(* CoDeSys 2.3 library: 3000ext.lib *)

(* Global variable list: Global_Constants *)
VAR_GLOBAL CONSTANT
(*CAN buses*)
	G_CANAPI_CAN1:BYTE := 0;
	G_CANAPI_CAN2:BYTE := 1;

(*Configuration flags*)
  	G_CANAPI_CFG_FLAGS_LISTEN_ONLY:WORD:=		16#0004;	(*CAN-interface is set to listen only mode*)

(*bit rates*)
	G_CANAPI_BAUDRATE_10K:WORD:= 	10;
	G_CANAPI_BAUDRATE_20K:WORD:= 	20;
	G_CANAPI_BAUDRATE_50K:WORD:= 	50;
	G_CANAPI_BAUDRATE_125K:WORD:= 	125;
	G_CANAPI_BAUDRATE_250K:WORD:= 	250;
	G_CANAPI_BAUDRATE_500K:WORD:= 	500;
	G_CANAPI_BAUDRATE_800K:WORD:= 	800;
	G_CANAPI_BAUDRATE_1000K:WORD:=1000;

(*protocols*)
	G_CANAPI_PROTOCOL_CANOPEN:BYTE := 0;
	G_CANAPI_PROTOCOL_ISOBUS:BYTE := 1;

END_VAR

(* Data type *)
TYPE CanApiBusConfiguration :
STRUCT
	i_enabled:WORD;			(* Used only internally. Variable is not needed in		*)
							(* function call CANAPI_INIT_BUS.						*)
	i_nbrOfInterface:WORD;	(* Number of the CAN channel channel(0,1,..)			*)
	i_bitRate:WORD;			(* CAN bitrate 											*)
	i_configFlags:WORD;		(* Configuration flags. See global contants				*)
END_STRUCT
END_TYPE

(* Data type *)
TYPE CanApiBusTimingParameters :
STRUCT
	i_nominalBitRate:DWORD;	(* CAN bitrate *)
	i_propSegment:WORD;		(* Propagation time segment (Tprop) *)
	i_phaseSegment1:WORD;	(* Phase buffer segment 1 (Tb1) *)
	i_phaseSegment2:WORD;	(* Phase buffer segment 2 (Tb2) *)
	i_sjw:WORD;					(* Resynchronization jump width (Tsjw) *)
	i_bitRateTolerance:WORD;	(*Allowed error in calculated bitRate.
									   Value in passed in 0.1 percent. So i.e. 15 means 1,5% *)
END_STRUCT
END_TYPE

(* Data type *)
TYPE CanApiMessage :
STRUCT
	id		: DWORD;				(*COB-ID of the message*)
	msgData	: ARRAY[0..7] OF BYTE;	(*Message data*)
	len		: BYTE;					(*Length of the message*)
END_STRUCT
END_TYPE

(* Data type *)
TYPE CanApiStatus :
STRUCT
	busOffCount		: DWORD;	(* Bus-Off error count *)
    ewarnCount		: DWORD;	(* EWarn Count *)

	txFifoOverruns	: DWORD;	(* Tx fifo overrun count *)
	txCount			: DWORD;	(* Tx message count *)
	txErrors		: DWORD;	(* Tx error count *)

	rxCount			: DWORD;	(* Rx message count *)
	rxErrors		: DWORD;   	(* Rx error count *)

	stuffErrCount	: DWORD;	(* Stuff error count *)
	formErrCount	: DWORD;	(* Form error count *)
	ackErrCount		: DWORD;	(* Ack error count *)
	bits1ErrCount	: DWORD;	(* Bits 1 error count *)
	bits0ErrCount	: DWORD;	(* Bits 0 error count *)
	crcErrCount		: DWORD;	(* CRC error count *)
END_STRUCT
END_TYPE

(* Data type *)
TYPE CommunicationParameters :
STRUCT
	CANChNR:WORD;	(* CAN channel number to use CoDeSys communication	*)
	kBitRate:WORD;	(* Communication bit rate of CAN					*)
	NodeID:WORD;	(* NodeID of CoDeSys Runtime						*)
	CableDetection:WORD;				(* Cable detection enabled/disabled	*)
	CableDetectionMask:WORD;			(* Mask bits for cable detection *)
	CableDetectionNodeOffset:WORD;		(* Node Id offset *)
	Termination:ARRAY [0..5] OF WORD;	(* CAN termination. *)
	CableDetectionPLCopenNodeIdOffset:WORD;
	Parameter:ARRAY [0..37] OF WORD;	(* Reserved for future use.
									This must fill structure's size to 126bytes(63 words)*)

	CAN1_NodeIdPLCopen:WORD;
	CAN1_kBitRate:WORD;
	CAN2_NodeIdPLCopen:WORD;
	CAN2_kBitRate:WORD;
	CAN3_NodeIdPLCopen:WORD;
	CAN3_kBitRate:WORD;
	CAN4_NodeIdPLCopen:WORD;
	CAN4_kBitRate:WORD;
	CAN5_NodeIdPLCopen:WORD;
	CAN5_kBitRate:WORD;
	CAN6_NodeIdPLCopen:WORD;
	CAN6_kBitRate:WORD;
END_STRUCT
END_TYPE

(* Data type *)
(* Contains information about HW assembly and software versions. *)
TYPE DeviceInfo :
STRUCT
	serialNumber 		: DWORD;	(* device serial number *)
 	deviceType			: WORD;		(* identifies device type: 3606, 3724... *)
 	boardRevision 		: WORD;		(* board revision A = 1, B = 2 ...*)
 	hwRevision 			: WORD;		(* HW revision *)
 	fwVersionMajor 		: WORD;		(* firmware major version number *)
 	fwVersionMinor 		: WORD;		(* firmware minor version number *)
 	piVersionMajor 		: WORD;		(* product info major version number *)
 	piVersionMinor 		: WORD;		(* product info minor version number *)
 	piExtVersionMajor 	: WORD;		(* extended product info major version number *)
 	piExtVersionMinor 	: WORD;		(* extended product info minor version number *)
 	bootVersionMajor 	: WORD;		(* boot major version number *)
 	bootVersionMinor 	: WORD;		(* boot minor version number *)
END_STRUCT
END_TYPE

(* Data type *)
TYPE DeviceInfoDate :
STRUCT
     fwVerDate:STRING(8);     (*< "mm/dd/yy" *)
     fwVerTime:STRING(8);     (*< "hh:mm:ss" *)
     piVerDate:STRING(8);     (*< "mm/dd/yy" *)
     piVerTime:STRING(8);     (*< "hh:mm:ss" *)
     piExtVerDate:STRING(8);  (*< "mm/dd/yy" *)
     piExtVerTime:STRING(8);  (*< "hh:mm:ss" *)
     bootVerDate:STRING(8);   (*< "mm/dd/yy" *)
     bootVerTime:STRING(8);   (*< "hh:mm:ss" *)
END_STRUCT
END_TYPE

(* Data type *)
TYPE ErrorLogEvent :
STRUCT
	timestamp : DWORD;  (* Error timestamp. RTC System TIME from boot. *)
	errorCode : INT;	(* Error code *)
	info 	  : DWORD;	(* Additional info *)
END_STRUCT
END_TYPE

(* Data type *)
TYPE IECVectors :
(
	INTCC16,			(* CAPCOM2 Request 16 *)
	INTCC17,			(* CAPCOM2 Request 17 *)
	INTCC18,			(* CAPCOM2 Request 18 *)
	INTCC19,			(* CAPCOM2 Request 19 *)
	INTCC20,			(* CAPCOM2 Request 20 *)
	INTCC21,			(* CAPCOM2 Request 21 *)
	INTCC22,			(* CAPCOM2 Request 22 *)
	INTCC23,			(* CAPCOM2 Request 23 *)
	INTCC24,			(* CAPCOM2 Request 24 *)
	INTCC25,			(* CAPCOM2 Request 25 *)
	INTCC26,			(* CAPCOM2 Request 26 *)
	INTCC27,			(* CAPCOM2 Request 27 *)
	INTCC28,			(* CAPCOM2 Request 28 *)
	INTCC29,			(* CAPCOM2 Request 29 *)
	INTCC30,			(* CAPCOM2 Request 30 *)
	INTCC31,			(* CAPCOM2 Request 31 *)
	INTT2,				(* GPT1 Timer 2 *)
	INTT3,				(* GPT1 Timer 3 *)
	INTT4,				(* GPT1 Timer 4 *)
	INTT5,				(* GPT1 Timer 5 *)
	INTT6,				(* GPT1 Timer 6 *)
	INTCR,			(* GPT2 CAPREL *)
	INTT7,				(* CAPCOM2 Timer 7 *)
	INTT8,				(* CAPCOM2 Timer 8 *)
	INTADC0,			(* A/D Converter Request 0 *)
	INTADC1,			(* A/D Converter Request 1 *)
	INTADC2,			(* A/D Converter Request 2 *)
	INTADC3,			(* A/D Converter Request 3 *)
	INTADC4,			(* A/D Converter Request 4 *)
	INTADC5,			(* A/D Converter Request 5 *)
	INTADC6,			(* A/D Converter Request 6 *)
	INTADC7,			(* A/D Converter Request 7 *)
	INTCCU60_0,		(* CCU60 Request 0 *)
	INTCCU60_1,		(* CCU60 Request 1 *)
	INTCCU60_2,		(* CCU60 Request 2 *)
	INTCCU60_3,		(* CCU60 Request 3 *)
	INTCCU61_0,		(* CCU61 Request 0 *)
	INTCCU61_1,		(* CCU61 Request 1 *)
	INTCCU61_2,		(* CCU61 Request 2 *)
	INTCCU61_3,		(* CCU61 Request 3 *)
	INTCCU62_0,		(* CCU62 Request 0 *)
	INTCCU62_1,		(* CCU62 Request 1 *)
	INTCCU62_2,		(* CCU62 Request 2 *)
	INTCCU62_3,		(* CCU62 Request 3 *)
	INTCCU63_0,		(* CCU63 Request 0 *)
	INTCCU63_1,		(* CCU63 Request 1 *)
	INTCCU63_2,		(* CCU63 Request 2 *)
	INTCCU63_3,		(* CCU63 Request 3 *)
	INTCAN0,			(* CAN0 *)
	INTCAN1,			(* CAN1 *)
	INTCAN2,			(* CAN2 *)
	INTCAN3,			(* CAN3 *)
	INTCAN4,			(* CAN4 *)
	INTCAN5,			(* CAN5 *)
	INTCAN6,			(* CAN6 *)
	INTCAN7,			(* CAN7 *)
	INTCCU0_T0,		(* CAPCOM1 Timer 0 Request *)
	INTCCU0_T1,		(* CAPCOM1 Timer 1 Request *)
	INTCC0,			(* CAPCOM1 Request 0 *)
	INTCC1,			(* CAPCOM1 Request 1 *)
	INTCC2,			(* CAPCOM1 Request 2 *)
	INTCC3,			(* CAPCOM1 Request 3 *)
	INTCC4,			(* CAPCOM1 Request 4 *)
	INTCC5,			(* CAPCOM1 Request 5 *)
	INTU0C0_0,		(* USIC0 CH0 SR0 *)
	INTU0C0_1,		(* USIC0 CH0 SR1 *)
	INTU0C0_2,		(* USIC0 CH0 SR2 *)
	INTU0C1_0,		(* USIC0 CH1 SR0 *)
	INTU0C1_1,		(* USIC0 CH1 SR1 *)
	INTU0C1_2,		(* USIC0 CH1 SR2 *)
	INTU1C0_0,		(* USIC1 CH0 SR0 *)
	INTU1C0_1,		(* USIC1 CH0 SR1 *)
	INTU1C0_2,		(* USIC1 CH0 SR2 *)
	INTU1C1_0,		(* USIC1 CH1 SR0 *)
	INTU1C1_1,		(* USIC1 CH1 SR1 *)
	INTU1C1_2,		(* USIC1 CH1 SR2 *)
	INTU2C0_0,		(* USIC2 CH0 SR0 *)
	INTU2C0_1,		(* USIC2 CH0 SR1 *)
	INTU2C0_2,		(* USIC2 CH0 SR2 *)
	INTU2C1_0,		(* USIC2 CH1 SR0 *)
	INTU2C1_1,		(* USIC2 CH1 SR1 *)
	INTU2C1_2,		(* USIC2 CH1 SR2 *)
	INTU3C0_0,		(* USIC3 CH0 SR0 *)
	INTU3C0_1,		(* USIC3 CH0 SR1 *)
	INTU3C0_2,		(* USIC3 CH0 SR2 *)
	INTU3C1_0,		(* USIC3 CH1 SR0 *)
	INTU3C1_1,		(* USIC3 CH1 SR1 *)
	INTU3C1_2,		(* USIC3 CH1 SR2 *)
	INTERU_0,		(* SCU External Request 0 *)
	INTERU_1,		(* SCU External Request 1 *)
	INTERU_2,		(* SCU External Request 2 *)
	INTSCU_1,		(* SCU Interrupt 1 *)
	INTSCU_0,		(* SCU Interrupt 0 *)
	INTERU_3,		(* SCU External Request 3 *)
	INTRTC,			(* RTC *)
	INTEOP,			(* End of PEC Subchannel *)
	INTCC6,			(* CAPCOM1 Request 6 *)
	INTCC7,			(* CAPCOM1 Request 7 *)
	INTCC8,			(* CAPCOM1 Request 8 *)
	INTCC9,			(* CAPCOM1 Request 9 *)
	INTCC10,			(* CAPCOM1 Request 10 *)
	INTCC11,			(* CAPCOM1 Request 11 *)
	INTCC12,			(* CAPCOM1 Request 12 *)
	INTCC13,			(* CAPCOM1 Request 13 *)
	INTCC14,			(* CAPCOM1 Request 14 *)
	INTCC15,			(* CAPCOM1 Request 15 *)
	INTU4C0_0,		(* USIC4 CH0 SR0 *)
	INTU4C0_1,		(* USIC4 CH0 SR1 *)
	INTU4C0_2,		(* USIC4 CH0 SR2 *)
	INTU4C1_0,		(* USIC4 CH1 SR0 *)
	INTU4C1_1,		(* USIC4 CH1 SR1 *)
	INTU4C1_2		(* USIC4 CH1 SR2 *)
);
END_TYPE

(* Data type *)
TYPE IoModes :
(
	IO_MODE_DISABLED,				(* Channel is disabled.							*)
	IO_PWFM_MODE_DIGITAL_OUTPUT,	(* Digital Out mode.*)
	IO_PWFM_MODE_DIRECT_PWFM,		(* Pulse width modulation mode. Pulse ratio is
											controlled from %Q area.				*)
	IO_PWFM_MODE_CURRENT_CONTROLLER,(* Not supported mode.							*)
	IO_PWFM_MODE_STEP_MOTOR,		(* Pulse amount is defined in PLCopen %Q area.	*)
	IO_PULSEIN_MODE_1CH,			(* One channel pulse input mode.				*)
	IO_PULSEIN_MODE_2CH,			(* Two channel pulse input mode.				*)
	IO_PULSEIN_MODE_RESET,			(* Channel is in reset mode.					*)
	IO_PULSEIN_MODE_2CH_DIR,		(* Two ch mode where 2nd ch defines direction.	*)
	IO_PULSEIN_MODE_FREQUENCY,		(* One channel mode, counts pulse frequency.	*)
	IO_PULSEIN_MODE_PULSEWIDTH,		(* One channel mode, counts pulse width.		*)
	IO_PULSEIN_MODE_DI				(* Channel is in Digital Input mode.			*)
);
END_TYPE

(* Data type *)
TYPE MEMORYDIMENSION :
STRUCT
	StartAdr:DWORD;	(* Beginning address of memory	*)
	EndAdr:DWORD;	(* Ending address of memory		*)
	Size:DWORD;		(* Length of memory in bytes	*)
END_STRUCT
END_TYPE

(* POU CANAPI_ADD_MO, ST *)
(*
----------------------------------------------------------
POU:													*)
FUNCTION CANAPI_ADD_MO : BYTE							(*
----------------------------------------------------------
Description:
	Function returns the message object number, 
	which is reserved to given channel.
	Unit has 255 message objects and runtime uses 0 & 1.
	If function returns 0 there are no more objects to use.
----------------------------------------------------------
*)
VAR_INPUT
	i_Channel:BYTE;	(* CAN channel(0,1,..). *)
END_VAR
VAR
END_VAR
;
END_FUNCTION

(* POU CANAPI_CHANGE_MO_COBID, ST *)
(*
----------------------------------------------------------
POU:													*)
FUNCTION CANAPI_CHANGE_MO_COBID : INT					(*
----------------------------------------------------------
Description:
	Function changes COBID from message object.

	Returns 0 after succesful operation.
----------------------------------------------------------
*)
VAR_INPUT
	i_Mo:BYTE;	(* Target message object *)
	i_Id:DWORD;	(* New COBID *)
END_VAR
VAR
END_VAR
;
END_FUNCTION

(* POU CANAPI_CHANGE_MO_MASK, ST *)
(*
-----------------------------------------------------------
POU:													*)
FUNCTION CANAPI_CHANGE_MO_MASK : INT					(*
----------------------------------------------------------
Description:
	Function changes mask from message object.

	Returns 0 after succesful operation.
----------------------------------------------------------
*)
VAR_INPUT
	i_Mo:BYTE;		(* Target message object *)
	i_Mask:DWORD;	(* New mask *)
END_VAR
VAR
END_VAR
;
END_FUNCTION

(* POU CANAPI_CHECK_NEW_MESSAGE, ST *)
(*
----------------------------------------------------------
POU:													*)
FUNCTION CANAPI_CHECK_NEW_MESSAGE : BYTE				(*
----------------------------------------------------------
Description:
	Function returns message object number that have new received message.
	Return 0 if there is no new messages.
----------------------------------------------------------
*)
VAR_INPUT
	i_Channel:BYTE;	(* CAN channel(0,1,..) that will be checked. *)
END_VAR
VAR
END_VAR
;
END_FUNCTION

(* POU CANAPI_CONFIGURE_MO, ST *)
(*
-----------------------------------------------------------
POU:													*)
FUNCTION CANAPI_CONFIGURE_MO : INT						(*
-----------------------------------------------------------
Description:
	Function configures given i_MO CAN message object.
	Only 1 transmit message object is allowed per channel.

	Function returns errorvalue or 0=Ok.
-----------------------------------------------------------
*)
VAR_INPUT
	i_ID:DWORD;			(* COB id Valid range 0..16#7FF for 11bit ID or*)
						(*16#20000000-16#3FFFFFFF for 29bit ID	*)
	i_MASK:DWORD;		(* COB mask	range same as above			*)
	i_DLC:BYTE;			(* Message length 0..8 bytes			*)
	i_MO:BYTE;			(* Object identity number 2..255		*)
END_VAR
VAR
END_VAR
;
END_FUNCTION

(* POU CANAPI_GET_STATUS, ST *)
(*
----------------------------------------------------------
POU:													*)
FUNCTION CANAPI_GET_STATUS : INT						(*
----------------------------------------------------------
Description:
	Gets structure CanApiStatus information from CAN.
	Return 0 after succesful operation.
----------------------------------------------------------
*)
VAR_INPUT
	i_Channel:BYTE;						(* CAN channel(0,1,..). *)
	i_Status:POINTER TO CanApiStatus; 	(* Pointer to status structure *)
END_VAR
VAR
END_VAR
;
END_FUNCTION

(* POU CANAPI_INIT_BUS, ST *)
(*
----------------------------------------------------------
POU:													*)
FUNCTION CANAPI_INIT_BUS : INT							(*
----------------------------------------------------------
Description:
	Function configures CAN interface.
	Function will return errorvalue or zero=no error.
----------------------------------------------------------
*)
VAR_INPUT
	i_Config: POINTER TO CanApiBusConfiguration; (* Pointer to configuration struct *)
END_VAR
VAR
END_VAR
;
END_FUNCTION

(* POU CANAPI_INIT_BUS_EXTENDED, ST *)
FUNCTION CANAPI_INIT_BUS_EXTENDED : INT			(*
----------------------------------------------------------
Description:
	Function configures CAN interface. This is called if non-standard CAN bus timing is used..
	Function will return errorvalue or zero=no error.
----------------------------------------------------------
----------------------------------------------------------
Version History:
	0.0.1	170217 MNN First Version
-----------------------------------------------------------
*)
VAR_INPUT
	i_Config: POINTER TO CanApiBusConfiguration; 		(* Pointer to configuration struct. NOTE: i_bitRate is unused while timing parameters are given in CanApiBusTimingParameters struct*)
	i_Timing: POINTER TO CanApiBusTimingParameters; (* Pointer to timingParameters struct *)
END_VAR
VAR
END_VAR
;
END_FUNCTION

(* POU CANAPI_INIT_SAMPLEPOINT, ST *)
FUNCTION CANAPI_INIT_SAMPLEPOINT : INT		(*
----------------------------------------------------------
Description:
Function selects protocol that is used with CAN interface. 
This is used to set ISOBUS samplepoint. CANopen doesn't need this function. 
This function must be called before CANAPI_INIT_BUS, otherwise the samplepoint is CANopen by default.
----------------------------------------------------------
Version History:
	0.0.1	170217 MNN First Version
-----------------------------------------------------------
*)
VAR_INPUT
	i_Channel:BYTE;			(* CAN channel (0,1,..). *)
	i_Protocol:BYTE;			(* CAN protocol (CANopen, ISOBUS,..) *)
END_VAR
VAR
END_VAR
;
END_FUNCTION

(* POU CANAPI_RECEIVE_MO, ST *)
(*
----------------------------------------------------------
POU:													*)
FUNCTION CANAPI_RECEIVE_MO : INT						(*
----------------------------------------------------------
Description:
	Read CAN-message from message object.

	Return 0 after succesful operation.
----------------------------------------------------------
*)
VAR_INPUT
	i_Mo:BYTE;						(* Message object *)
	i_Msg:POINTER TO CanApiMessage;	(* Pointer to CanApisMessage *)
END_VAR
VAR
END_VAR
;
END_FUNCTION

(* POU CANAPI_REMOVE_ALL_MOS, ST *)
(*
----------------------------------------------------------
POU:													*)
FUNCTION CANAPI_REMOVE_ALL_MOS : INT					(*
----------------------------------------------------------
Description:
	Remove all registered message objects from all CAN-channels.

	Return 0 after succesful operation.
----------------------------------------------------------
*)
VAR_INPUT
END_VAR
VAR
END_VAR
;
END_FUNCTION

(* POU CANAPI_REMOVE_MOS, ST *)
(*
----------------------------------------------------------
POU:													*)
FUNCTION CANAPI_REMOVE_MOS : INT						(*
----------------------------------------------------------
Description:
	Remove all registered message objects.

	Return 0 after succesful operation.
----------------------------------------------------------
*)
VAR_INPUT
	i_Channel:BYTE;	(* CAN channel(0,1,..). *)
END_VAR
VAR
END_VAR
;
END_FUNCTION

(* POU CANAPI_SEND, ST *)
(*
----------------------------------------------------------
POU:													*)
FUNCTION CANAPI_SEND : INT								(*
----------------------------------------------------------
Description:
	Send message. 
	Send buffer must be set before using send.

	Return 0 after succesful operation.
----------------------------------------------------------
*)
VAR_INPUT
	i_Channel:BYTE;					(* CAN channel(0,1,..). *)
	i_Msg:POINTER TO CanApiMessage;	(* Pointer to CanApiMessage *)
END_VAR
VAR
END_VAR
;
END_FUNCTION

(* POU CANAPI_SET_SEND_BUFFER, ST *)
(*
----------------------------------------------------------
POU:													*)
FUNCTION CANAPI_SET_SEND_BUFFER : INT					(*
----------------------------------------------------------
Description:
	Set send buffer. Sets IEC allocated transmit buffer to 
	runtime CAN-transmit system.

	Return 0 after succesful operation.
----------------------------------------------------------
*)
VAR_INPUT
	i_Channel:BYTE;			(* CAN channel(0,1,..). *)
	i_BufferSize:WORD;		(* Number of CanApiMessage in buffer *)
	i_BufferPointer:POINTER TO CanApiMessage; (* Pointer to buffer *)
END_VAR
VAR
END_VAR
;
END_FUNCTION

(* POU COMMPARAMSGET, ST *)
(*
-----------------------------------------------------------
POU:													*)
FUNCTION COMMPARAMSGET : INT							(*
-----------------------------------------------------------
Description:
Function reads CommunicationParameters struct from firmware.
return Firmware error code.
-----------------------------------------------------------
Version History:
	0.0.1	120612 PasiM First Version
-----------------------------------------------------------
*)
VAR_INPUT
	i_Address:POINTER TO CommunicationParameters;	(* CommunicationParameters struct *)
													(* where to load parameters. 	  *)
END_VAR
VAR
END_VAR
;
END_FUNCTION

(* POU COMMPARAMSSET, ST *)
(*
-----------------------------------------------------------
POU:													*)
FUNCTION COMMPARAMSSET : INT							(*
-----------------------------------------------------------
Description:
Function writes CommunicationParameters struct to firmware.
return Firmware error code.	
-----------------------------------------------------------
Version History:
	0.0.1	120612 PasiM First Version
-----------------------------------------------------------
*)
VAR_INPUT
	i_Address:POINTER TO CommunicationParameters;(* CommunicationParameters struct to save. *)
END_VAR
VAR
END_VAR
;
END_FUNCTION

(* POU COMMPARAMSSETWAIT, ST *)
(*
-----------------------------------------------------------
POU:													*)
FUNCTION COMMPARAMSSETWAIT : BOOL(*
-----------------------------------------------------------
Description:
Function sets inhibitime for communication parameters write 
to flash memory. System default wait time is 100s.
-----------------------------------------------------------
Version History:
	0.0.1	120831 PasiM First Version
-----------------------------------------------------------
*)
VAR_INPUT
	i_Seconds:WORD;(*Write inhibit time in seconds*)
END_VAR
VAR
END_VAR
;
END_FUNCTION

(* POU DATAPARAMSGET, ST *)
(*
-----------------------------------------------------------
POU:													*)
FUNCTION DATAPARAMSGET : INT							(*
-----------------------------------------------------------
Description:
Function copies parameters from Parameter FLASH to PLCopen memory. Parameter
Array length is 63 * 16bit = 126 bytes. 
i_Address is Pointer to PLCopen memory that contains 63*16bit variables. 
return Firmware error code.
	
-----------------------------------------------------------
Version History:
	0.0.1	120612 PasiM First Version
-----------------------------------------------------------
*)
VAR_INPUT
	i_Address:DWORD; (* Pointer to PLCopen memory that contains 63*16bit variables. *)
END_VAR
VAR
END_VAR
;
END_FUNCTION

(* POU DATAPARAMSSET, ST *)
(*
-----------------------------------------------------------
POU:													*)
FUNCTION DATAPARAMSSET : INT							(*
-----------------------------------------------------------
Description:
Function copies parameters from PLCopen memory to the Parameter FLASH. 
One parameter block length is 63 * 16bit = 126 bytes. 
i_Address is Pointer to 63 * 16bit data what will be stored to FLASH.
return Firmware error code.	
-----------------------------------------------------------
Version History:
	0.0.1	120612 PasiM First Version
-----------------------------------------------------------
*)
VAR_INPUT
	i_Address:DWORD; (* Pointer to 63 * 16bit data what will be stored to FLASH. *)
END_VAR
VAR
END_VAR
;
END_FUNCTION

(* POU DATAPARAMSSETWAIT, ST *)
(*
-----------------------------------------------------------
POU:													*)
FUNCTION DATAPARAMSSETWAIT : BOOL(*
-----------------------------------------------------------
Description:
Function sets inhibitime for system parameters write 
to flash memory. System default wait time is 100s.
-----------------------------------------------------------
Version History:
	0.0.1	120831 PasiM First Version
-----------------------------------------------------------
*)
VAR_INPUT
	i_Seconds:WORD;(*Write inhibit time in seconds*)
END_VAR
VAR
END_VAR
;
END_FUNCTION

(* POU IEC_READ_INPUTS, ST *)
FUNCTION IEC_READ_INPUTS : INT		(*
----------------------------------------------------------
Description:
Function calls runtime to update current input states from HW to %IW variables.
----------------------------------------------------------
Version History:
	0.0.1	170217 MNN First Version
-----------------------------------------------------------
*)
VAR_INPUT
END_VAR
VAR
END_VAR
;
END_FUNCTION

(* POU IEC_WRITE_OUTPUTS, ST *)
FUNCTION IEC_WRITE_OUTPUTS : INT		(*
----------------------------------------------------------
Description:
Function calls runtime to update current outputs from %QW variables to HW.
----------------------------------------------------------
Version History:
	0.0.1	170217 MNN First Version
-----------------------------------------------------------
*)
VAR_INPUT
END_VAR
VAR
END_VAR
;
END_FUNCTION

(* POU IO_PULSEIN_RESET, ST *)
(*
--------------------------------------------------------------------------------
POU:																		  *)
FUNCTION IO_PULSEIN_RESET : INT

(*
--------------------------------------------------------------------------------
Description:

Reset Pulse Input channel pulse counter value and measurement data. 
Channel pulse counter value is set new value defined by i_ResetValue.
Channel alternative measurement data value (frequency or pulse width) is set to 
zero.  

Return value is error code. 0 = OK.

--------------------------------------------------------------------------------
Version History:
	0.0.1	130612 JuhaO 	Initial version
--------------------------------------------------------------------------------
*)

VAR_INPUT
	i_ChannelNbr:WORD;	(* 	Pulse input channel number. *)
	i_ResetValue:WORD;	(* 	Reset value for pulse counter. *)
END_VAR
VAR
END_VAR
;
END_FUNCTION

(* POU IO_PULSEIN_SET_CONFIG, ST *)
(*
-----------------------------------------------------------
POU:													*)
FUNCTION IO_PULSEIN_SET_CONFIG : INT					(*
-----------------------------------------------------------
Description:
	Defines usage of pulseinput channel.
	Function returns errorvalue or 0.
	IO_PULSEIN_MODE_1CH
		In 1channel mode pulsechannel will count pulses from one pulseinput to IW 
		memory.
	IO_PULSEIN_MODE_2CH
		In 2ch mode function i_ChannelPairNbr input will tell the B channel of 
		quatrature input.
	IO_PULSEIN_MODE_RESET
		Function input i_ResetChnNbr is channel which will be reseted. Used as Z 
		pulseinput.
	IO_PULSEIN_MODE_2CH_DIR
		2 channel mode where ChannelPair will be counting direction.
	IO_PULSEIN_MODE_FREQUENCY
		In frequency mode pulsechannel will count frequency from one pulseinput to IW 
		memory.
	IO_PULSEIN_MODE_PULSEWIDTH
		In pulsewidth measurement mode pulsechannel will measure incomming pulses 
		hightime in microseconds to IW memory.
	IO_PULSEIN_MODE_DI
		In digital input mode pulsechannel will give digital state from one pulseinput 
		to IW memory.
-----------------------------------------------------------
Version History:
	0.0.1	120611 PasiM First Version
	0.0.2	130405 JuhaO Added input param iGateTime.
-----------------------------------------------------------
*)
VAR_INPUT
	i_Mode:IoModes;						(* 	Used mode for pulse input channel. 												*)
	i_ChannelNbr:WORD;					(* 	Pulse input channel number which is configured. 								*)
	i_ResetChnNbr:BYTE;					(* 	Number of reseted channel. Valid only if reset channel mode is chosen. 			*)
	i_ChannelPairNbr:BYTE;				(* 	Digitalinput number of channel pair. Valid only if two channel mode is chosen.	*)
	i_EdgeSelect:BYTE;					(* 	Selects edge type for pulse input. 0 - Count one edge , 1 - Count both edges. 	*)
	i_EdgePolarity:BYTE;				(* 	Selects polarity for edge counting. 0 - Rising edge , 1 - Falling edge. 		*)
	i_GateTime:WORD;					(*  Measurement gate time in milliseconds.											*)
END_VAR
VAR
END_VAR
;
END_FUNCTION

(* POU IO_PWFM_SET_CONFIG, ST *)
FUNCTION IO_PWFM_SET_CONFIG : INT

(*
	Function is used to set configuration for pwfm channel.
	Pwfm channel can be in different modes depending hardware. Check technical manual 
	for detailed information about possible modes.
	Firmware protect wrong usage. 
	If user tries to use channel in wrong mode function gives error code and sets 
	channel to disabled mode. 

	Below is listed which configuration parameters are valid in different modes.

						Digital Output		Direct Pwfm		Step Motor
	pwfmMode			X					X				X					
	pwfmChn				X					X				X					
	

	Pwfm channel can be used following modes:

	IO_PWFM_MODE_DISABLED
		Pwfm channel is disabled and output is always set to off state.		

	IO_PWFM_MODE_DIGITAL_OUTPUT
		Pwfm channel is used as digital output and user use boolean variable 
		o_PwfmChnX_DoState	set wanted output state.

	IO_PWFM_MODE_DIRECT_PWFM
		In direct pwfm mode user can set pulse ratio and frequency for pwfm channel. 
		In low frequencies user must notice that channel executes always one pulse 
		after new values are used. 
		This means for example in 10Hz frequency that new values are taken in use 
		after 100ms.

	IO_PWFM_MODE_STEP_MOTOR
		In step motor mode user sets number of wanted pulses which channel generates. 
		Width and frequency can be set through normal output variables in plc configuration.

	Version info:
	0.01	
		23.03.2011	Mika Lammila		First version
		31.01.2011	Mika Lammila	
	0.02
		120807	Pasi Myllymäki Changes for 3000 series.	
*)

VAR_INPUT
	i_PwfmMode:IoModes;	(* Used mode *)
	i_PwfmChn:WORD;		(* Pwfm channel *)
END_VAR
VAR
END_VAR
;
END_FUNCTION

(* POU IO_SET_AI_BUFFER, ST *)
(*
-----------------------------------------------------------
POU:													*)
FUNCTION_BLOCK IO_SET_AI_BUFFER							(*
-----------------------------------------------------------
Description:
	Defines ringbuffer of analog measuremests for 
	analog input channel
	
-----------------------------------------------------------
Version History:
	0.0.1	120611 PasiM First Version	
-----------------------------------------------------------
*)
VAR_INPUT
	i_CH:WORD;		(* Channel [0..XX]											*)
	i_Data:POINTER TO WORD;	(* Address of buffer (use ADR operator) use even pointers
						for word alingment										*)
	i_Length:WORD;	(* Buffer length in bytes (use SIZEOF operator).
						Length must be divisible by 2							*)
END_VAR
VAR_OUTPUT
	o_Write:WORD;	(* Position of last value in ringbuffer *)
END_VAR
VAR
END_VAR
;
END_FUNCTION_BLOCK

(* POU IO_SET_LED, ST *)
(*
-----------------------------------------------------------
POU:													*)
FUNCTION IO_SET_LED : INT								(*
-----------------------------------------------------------
Description:
	Function is used to set status led. User sets boolean inputs as needed and 
	firmware controls output led.
	Function returns Errorcode or 0.
	Function controls status LED (if exsists) according to application status. 
	LED is also controlled by HW and FW. LED's control priority order is following 
	1. HW, 2. FW, 3. Application. (application has the lowest priority).

	i_SystemOk 	i_RunWithErrors 	i_InitState 	GreenLed	RedLed
	X			X					T				ON			OFF
 	T			F					F				Blink 2 Hz	OFF
	T			T					F				OFF			Blink 5 Hz
	F			X					F				OFF			Blink 2 Hz
 

-----------------------------------------------------------
Version History:
	0.0.1	120611 PasiM First Version
-----------------------------------------------------------
*)
VAR_INPUT
	i_SystemOk:		BOOL;(* System OK information from application 					*)
	i_RunWithErrors:BOOL;(* HW/SW error information from application (for example 	*)
						 (* short circuit in output)								*)
 	i_InitState: 	BOOL;(* True until application initializing functions are done	*)
END_VAR
VAR
END_VAR
;
END_FUNCTION

(* POU LOG_ERROR, ST *)
(*
This function adds an error with timestamp to SBRAM log.

Return values:
FwOk					Error added successfully to log.
FwPLCopenErrorWrong		Given i_ErrorCode too small (i.e. less than 10000).

*)
FUNCTION LOG_ERROR : INT
VAR_INPUT
	i_ErrorCode : INT;		(* Application error code *)
	i_Info		: DWORD;	(* Additional information *)

END_VAR
VAR
END_VAR
;
END_FUNCTION

(* POU LOG_GET_EVENT, ST *)
(*
This function reads an error from log.
Reading starts from the beginning of SBRAM.
Each call return the next logged error.

When all errors are read, return value is FwErrorLogEnd, 
and read pointer is set back to the beginning of SBRAM.


Return values:
FwOk						Error read ok.
FwErrorGetLogParameterNull	Null event pointer given.
FwErrorLogEnd				End of log reached.
FwSbRamEnd 					Read reach the end of the SBRAM. Data copied to dest may be 
							shorter than len defines.
FwSbRamReadPtr				Internal read index is out of range.
	

*)
FUNCTION LOG_GET_EVENT : INT
VAR_INPUT
	i_Event : POINTER TO ErrorLogEvent;

END_VAR
VAR
END_VAR
;
END_FUNCTION

(* POU NVRAMCOPY, ST *)
(*
-----------------------------------------------------------
POU:													*)
FUNCTION_BLOCK NVRAMCOPY                                (*
-----------------------------------------------------------
Description:
Function copyes data from/to nonvolatile RAM to user RAM.

i_Enable	Rising edge: the function block starts the action.
i_DestAdr 	Destination address of copy.
i_SrcAdr 	Source address of copy.
i_Length 	Amount of data in bytes.

o_Done		TRUE indicates that the function block has completed processing.
o_Busy		TRUE indicates that the FUNCTION block is still processing.
o_Error		TRUE indicates that an error has occurred.
o_ErrorId	Error number


-----------------------------------------------------------
Version History:
	0.0.1	120612 PasiM First Version
-----------------------------------------------------------
*)
VAR_INPUT
	i_Enable:BOOL;	(* Rising edge: the function block starts the action. *)
	i_DestAdr:DWORD;(* Destination address of copy. *)
	i_SrcAdr:DWORD;	(* Source address of copy. *)
	i_Length:DWORD; (* Amount of data in bytes. *)
END_VAR
VAR_OUTPUT
	o_Done:BOOL;	(* TRUE indicates that the function block has completed processing. *)
	o_Busy:BOOL;	(* TRUE indicates that the function block is still processing. *)
	o_Error:BOOL;	(* TRUE indicates that an error has occurred. *)
	o_ErrorId:WORD;	(* Error number *)
END_VAR
VAR
END_VAR
;
END_FUNCTION_BLOCK

(* POU NVRAMGETSIZE, ST *)
(*
-----------------------------------------------------------
POU:													*)
FUNCTION NVRAMGETSIZE : DWORD							(*
-----------------------------------------------------------
Description:
Function fetces dimensions of nonvolatile memory.
Function returns size of nonvolatile RAM.
-----------------------------------------------------------
Version History:
	0.0.1	120612 PasiM First Version
-----------------------------------------------------------
*)
VAR_INPUT
	i_MemDAdr:POINTER TO MEMORYDIMENSION;(* Pointer to NVRAM memrodimensions struct. *)
END_VAR
VAR
END_VAR
;
END_FUNCTION

(* POU SYSINSTALLHANDLER, ST *)
FUNCTION SYSINSTALLHANDLER : INT	(*
----------------------------------------------------------
Description:
Re-directs interrupthandler from runtime to IEC-function.
----------------------------------------------------------
*)
VAR_INPUT
	i_Vector:WORD;		(* Index of interrupt vector *)
	i_POU:WORD;		(* Index of POU to call *)
END_VAR
VAR
END_VAR
;
END_FUNCTION

(* POU SYSTEM_CALL_POU, ST *)
(*
-----------------------------------------------------------
POU:													*)
FUNCTION SYSTEM_CALL_POU : BOOL								(*
-----------------------------------------------------------
Description:
Function calls POU with given POU number, use INDEXOF() operator
to get index of POU.
-----------------------------------------------------------
Version History:
	0.0.1	120831 PasiM First Version
-----------------------------------------------------------
*)
VAR_INPUT
	i_POU:WORD;	(*Index of POU to call*)
END_VAR
VAR
END_VAR
;
END_FUNCTION

(* POU SYSTEM_RESTART_PLCOPEN_APP, ST *)
(*
-----------------------------------------------------------
POU:													*)
FUNCTION SYSTEM_RESTART_PLCOPEN_APP : INT

(*
-----------------------------------------------------------
Description:
This function restarts the PLCopen Application. 
As input to function is given wanted reset action.
Function returns an error code.

-----------------------------------------------------------
Version History:
	0.0.1	120831 PasiM First Version
	0.0.2	130506 JuhaO iResetMode parameter and returnvalue
-----------------------------------------------------------
*)
VAR_INPUT
	i_ResetMode:BYTE; 	(* 	0 - Reset
							1 - Reset (Cold)
							2 - Reset (Original)
						*)
END_VAR
VAR
END_VAR
;
END_FUNCTION
